(*
JobNode manages the state of a job and it's execution.
*)
INTERFACE I_JobNode EXTENDS I_JobNodeInternal

(*
Notifies scheduler to aboort this job.
Returns Err.IncArg on State = Idle
*)
METHOD Abort : Result
VAR_INPUT
END_VAR
END_METHOD

(*
Starts the job and adds it to Workers queue.
Returns Err.IncArg on State <> Idle.
Returns Err.Itf0 on Worker = 0.
*)
METHOD Start : Result
VAR_INPUT
END_VAR
END_METHOD

END_INTERFACE

(* stored: Version 1.1.0.1
   Itf I_JobNode: Id {d740f790-ee67-445b-9a56-dbf77aaa8b7e}
   Method Abort: Id {bba4b53e-67ed-4af8-a6e2-ec322380ef7d}
   Method Start: Id {efd62966-8b23-4509-9c23-13ebf675ee3d} *)
